FUNCTION_BLOCK T_RoboConnect_SetToolAnalogOutput_CorrectIndexPasses EXTENDS T_UnitTestBase
VAR
  robot : I_RoboConnect;
  targetDO : UINT;
  myTestState, prevState :
    (INIT, ARRANGE, ACT, ASSERT) := INIT;
  expected, actual : BOOL;
  counter : UINT;
END_VAR

CASE myTestState OF
  INIT:
    StateChanged();
    myTestState := ARRANGE;

  ARRANGE:
    IF StateChanged() THEN
      expected := TRUE;
      robot.Connect();
    END_IF

    IF robot.Connected THEN
      myTestState := ACT;
    END_IF

  ACT:
    actual := robot.SetToolAnalogOutput(targetDO, 0.5);
    myTestState := ASSERT;

  ASSERT:
    assertion.AssertEquals_BOOL(expected, actual, 'actual := robot.SetToolAnalogOutput(targetDO, TRUE)');
    TestFinished();
    myTestState := INIT;

END_CASE

METHOD FB_init : BOOL
VAR_INPUT
  bInitRetains : BOOL; // if TRUE, the retain variables are initialized (warm start / cold start)
  bInCopyCode : BOOL; // if TRUE, the instance afterwards gets moved into the copy code (online change)
  TestSuite : tcl_SimpleUnitTestLibrary.I_TestSuite;
  robot : I_TcRobot;
  targetDo : UINT;
END_VAR
THIS^.robot := robot;
THIS^.targetDo := targetDo;
END_METHOD

METHOD PRIVATE StateChanged : BOOL
IF  myTestState = prevState THEN
  RETURN;
END_IF

prevState := myTestState;
StateChanged := TRUE;
END_METHOD

METHOD WaitForCycles : BOOL
VAR_INPUT
  maxCount : UINT;
END_VAR
counter := counter + 1;

IF counter = maxCount THEN
  counter := 0;
  WaitForCycles := TRUE;
END_IF
END_METHOD

END_FUNCTION_BLOCK

(* stored: Version 1.1.0.1
   POU T_TcRobot_SetToolAnalogOutput_CorrectIndexPasses: Id {3a640e89-adb0-40d3-a409-05fae6ac696e}, SpecialFunc None
   Method FB_init: Id {16f7c8de-595b-4dd2-b44c-29443dd93960}
   Method StateChanged: Id {ba5c73ff-28a2-42e8-9b30-1802081dca0d}
   Method WaitForCycles: Id {731a07fd-2e05-4453-9e17-68eed708c996} *)
